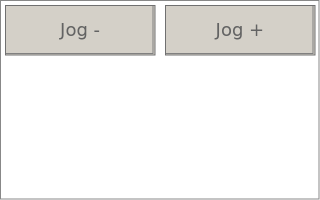
VISUALIZATION SingleAxisJogStandardSlow  // 320x200
VAR_IN_OUT
	btnJogPositive	: BOOL;
	btnJogNegative	: BOOL;
END_VAR
    Button (5,5 150x50), "Jog -"
        tap btnJogNegative
    Button (165,5 150x50), "Jog +"
        tap btnJogPositive
END_VISUALIZATION

(* stored: Version 1.1.0.1, ProductVersion 3.1.4024.9
   Visu SingleAxisJogStandardSlow: Id {5c7c93b6-a143-4214-b4b1-060fe67f97e3} *)
